// TIA Portal V17 export
// export: Created 2022-07-20T07:02:33.3488403Z, ExportSetting WithDefaults, DisplayName Totally Integrated Automation Portal, DisplayVersion V17, DisplayName TIA Portal Openness, DisplayVersion V17, DisplayName TIA Portal Version Control Interface, DisplayVersion V17, DisplayName SINAMICS Startdrive Advanced, DisplayVersion V17, DisplayName SINAMICS Startdrive G130, G150, S120, S150, SINAMICS MV, S210, DisplayVersion V17, DisplayName SINAMICS Startdrive G110M, G120, G120C, G120D, G120P, G115D, DisplayVersion V17, DisplayName STEP 7 Professional, DisplayVersion V17, DisplayName STEP 7 Safety, DisplayVersion V17, DisplayName WinCC Advanced, DisplayVersion V17
FUNCTION_BLOCK "FB10130_SMC_LC3F2"   // FB10130, LAD
{ S7_Optimized_Access := 'TRUE' }
VERSION : 0.1
// stored: AutoNumber false, IsIECCheckEnabled false, IsRetainMemResEnabled false, MemoryReserve 100, SetENOAutomatically false, UDAEnableTagReadback false
   VAR_INPUT
      Request_DownPosition : Bool;
      Request_UpPosition : Bool;
      Request_LimitForce : Bool;
      InvertDirection : Bool;
   END_VAR
   VAR_OUTPUT
      On : Bool;
      Set : Bool;
      "A-Phase" : Bool;
      States : "stSMCLC3F2States";
   END_VAR
BEGIN

REGION Network 1: Power activation 100%
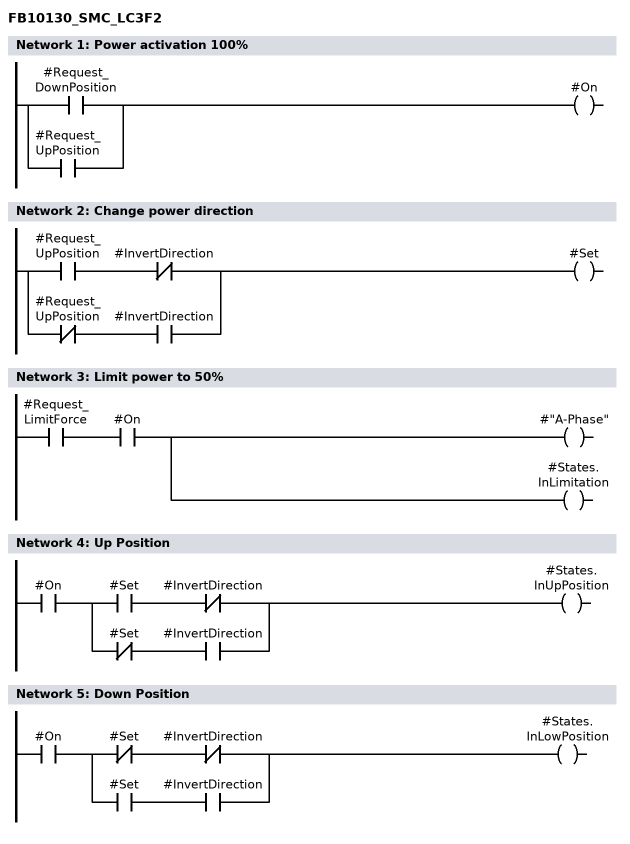
   RUNG wire#powerrail
      Contact( #Request_DownPosition )
      wire#w1
      Coil( #On )
   END_RUNG
   RUNG wire#powerrail
      Contact( #Request_UpPosition )
   END_RUNG wire#w1
   // the same network as SCL:
   #On := #Request_DownPosition OR #Request_UpPosition;
END_REGION

REGION Network 2: Change power direction
   RUNG wire#powerrail
      Contact( #Request_UpPosition )
      I_Contact( #InvertDirection )
      wire#w1
      Coil( #Set )
   END_RUNG
   RUNG wire#powerrail
      I_Contact( #Request_UpPosition )
      Contact( #InvertDirection )
   END_RUNG wire#w1
   // the same network as SCL:
   #Set := (#Request_UpPosition AND NOT #InvertDirection) OR (NOT #Request_UpPosition AND #InvertDirection);
END_REGION

REGION Network 3: Limit power to 50%
   RUNG wire#powerrail
      Contact( #Request_LimitForce )
      Contact( #On )
      wire#w1
      Coil( #"A-Phase" )
   END_RUNG
   RUNG wire#w1
      Coil( #States.InLimitation )
   END_RUNG
   // the same network as SCL:
   #"A-Phase" := #Request_LimitForce AND #On;
   #States.InLimitation := #"A-Phase";
END_REGION

REGION Network 4: Up Position
   RUNG wire#powerrail
      Contact( #On )
      wire#w1
      Contact( #Set )
      I_Contact( #InvertDirection )
      wire#w2
      Coil( #States.InUpPosition )
   END_RUNG
   RUNG wire#w1
      I_Contact( #Set )
      Contact( #InvertDirection )
   END_RUNG wire#w2
   // the same network as SCL:
   #States.InUpPosition := #On AND ((#Set AND NOT #InvertDirection) OR (NOT #Set AND #InvertDirection));
END_REGION

REGION Network 5: Down Position
   RUNG wire#powerrail
      Contact( #On )
      wire#w1
      I_Contact( #Set )
      I_Contact( #InvertDirection )
      wire#w2
      Coil( #States.InLowPosition )
   END_RUNG
   RUNG wire#w1
      Contact( #Set )
      Contact( #InvertDirection )
   END_RUNG wire#w2
   // the same network as SCL:
   #States.InLowPosition := #On AND ((NOT #Set AND NOT #InvertDirection) OR (#Set AND #InvertDirection));
END_REGION
END_FUNCTION_BLOCK
